{attribute 'GeneratedUsingTerminal: EL3201-0000-0016'}
{attribute addProperty BoxType "EL3201-0000-0016"}
{attribute addProperty Description "EL3201 1Ch. Ana. Input PT100 (RTD)"}
{attribute addProperty Physics "KK"}
{attribute addProperty Id "RTD_InputsAT %I*RTD_Inputs_EA9DF21E9WcStateAT %I*WcState_9091E0EB2InfoDataAT %I*InfoData_32EB74EA10"}
{attribute addProperty CRC "1997624545"}
{attribute addProperty Size "21"}
TYPE EL3201_771154E1 EXTENDS EtcSlaveTerminalBase_947E5A46 :
STRUCT
	{attribute addProperty Name "RTD_Inputs"}
	RTD_Inputs : RTD_Inputs_EA9DF21E;
	{attribute addProperty Name "WcState"}
	WcState : WcState_9091E0EB;
	{attribute addProperty Name "InfoData"}
	InfoData : InfoData_32EB74EA;
END_STRUCT
END_TYPE

(* stored: Version 1.2.0.0, ProductVersion 3.1.4024.9
   DUT EL3201_771154E1: Id {f0d534b6-cccf-40ac-a9a4-7b3b6d596f38} *)
